(* Schneider Machine Expert - Basic project 3 SW , 2Lamp, file version 1.8.0.0 *)
(* ProjectInformations: Name=New project *)

HARDWARE
  Cpu 0: TM221CE16R
  EthernetConfiguration: NetworkName=M221, IpAllocationMode=FixedAddress, IpAddress=0.0.0.0, SubnetMask=0.0.0.0
  SerialLineConfiguration: Baud=Baud19200, Parity=ParityEven, DataBits=DataBits8, StopBits=StopBits1, PhysicalMedium=PhysicalMediumRs485, TransmissionMode=TransmissionModeModbusRtu, SlaveId=1, Addressing=SlaveAddressing
  MastTask: UsePeriodScanMode=false, PeriodScan=100
  FastTask: Period=255
  CpuBehavior: StartingMode=StartAsPreviousState, AutoSaveRamOnEeprom=true, WatchdogPeriod=250

SYMBOLS  (address, symbol, comment, settings)

POU New POU
  (* SectionNumber=0 *)

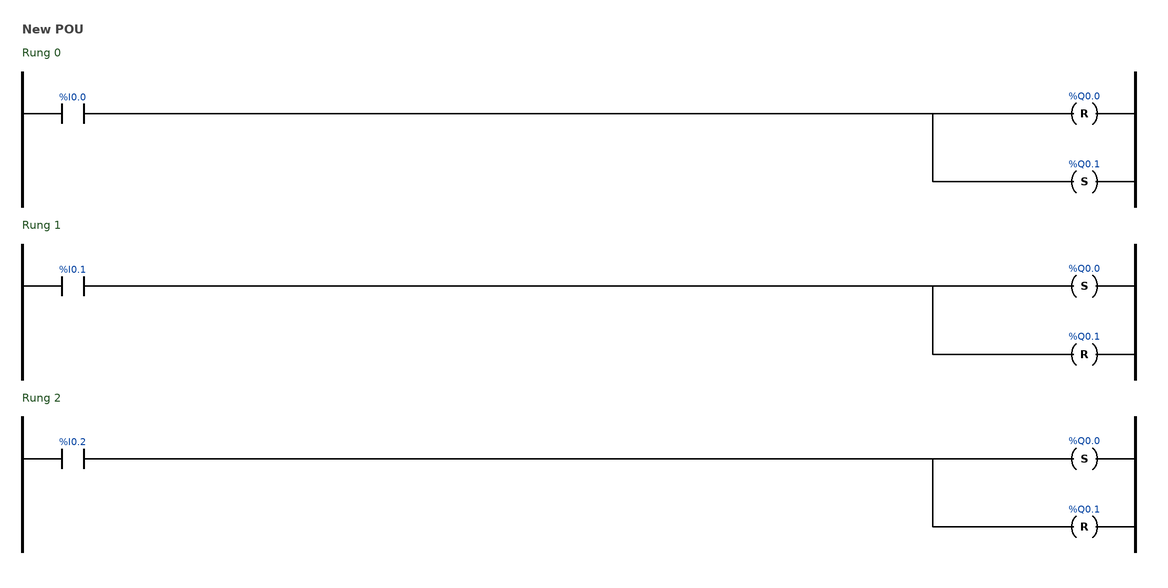

// Rung 0
  LD %I0.0
  R %Q0.0
  S %Q0.1
  // as ST:
  //   IF %I0.0 THEN %Q0.0 := FALSE; END_IF;
  //   IF %I0.0 THEN %Q0.1 := TRUE; END_IF;

// Rung 1
  LD %I0.1
  S %Q0.0
  R %Q0.1
  // as ST:
  //   IF %I0.1 THEN %Q0.0 := TRUE; END_IF;
  //   IF %I0.1 THEN %Q0.1 := FALSE; END_IF;

// Rung 2
  LD %I0.2
  S %Q0.0
  R %Q0.1
  // as ST:
  //   IF %I0.2 THEN %Q0.0 := TRUE; END_IF;
  //   IF %I0.2 THEN %Q0.1 := FALSE; END_IF;
